FUNCTION F_Inc : BOOL
VAR_INPUT
    in : ANY_INT;
END_VAR
VAR
    pSINT  : POINTER TO SINT;
    pINT   : POINTER TO INT;
    pDINT  : POINTER TO DINT;
    pLINT  : POINTER TO LINT;
    pUSINT : POINTER TO USINT;
    pUINT  : POINTER TO UINT;
    pUDINT : POINTER TO UDINT;
    pULINT : POINTER TO ULINT;
    pBYTE  : POINTER TO BYTE;
    pWORD  : POINTER TO WORD;
    pDWORD : POINTER TO DWORD;
END_VAR

CASE in.TypeClass OF
    __SYSTEM.TYPE_CLASS.TYPE_SINT:
        pSINT  := in.pValue;
        pSint^ := pSint^ + 1;

    __SYSTEM.TYPE_CLASS.TYPE_INT:
        pINT  := in.pValue;
        pINT^ := pINT^ + 1;

    __SYSTEM.TYPE_CLASS.TYPE_DINT:
        pDINT  := in.pValue;
        pDINT^ := pDINT^ + 1;

    __SYSTEM.TYPE_CLASS.TYPE_LINT:
        pLINT  := in.pValue;
        pLINT^ := pLINT^ + 1;

    __SYSTEM.TYPE_CLASS.TYPE_USINT:
        pUSINT  := in.pValue;
        pUSINT^ := pUSINT^ + 1;

    __SYSTEM.TYPE_CLASS.TYPE_UINT:
        pUINT  := in.pValue;
        pUINT^ := pUINT^ + 1;

    __SYSTEM.TYPE_CLASS.TYPE_UDINT:
        pUDINT  := in.pValue;
        pUDINT^ := pUDINT^ + 1;

    __SYSTEM.TYPE_CLASS.TYPE_ULINT:
        pULINT  := in.pValue;
        pULINT^ := pULINT^ + 1;
		
    __SYSTEM.TYPE_CLASS.TYPE_BYTE:
        pBYTE  := in.pValue;
        pBYTE^ := pBYTE^ + 1;
		
    __SYSTEM.TYPE_CLASS.TYPE_WORD:
        pWORD  := in.pValue;
        pWORD^ := pWORD^ + 1;
		
    __SYSTEM.TYPE_CLASS.TYPE_DWORD:
        pDWORD  := in.pValue;
        pDWORD^ := pDWORD^ + 1;
		
		
END_CASE

END_FUNCTION

(* stored: Version 1.1.0.1, ProductVersion 3.1.4024.12
   POU F_Inc: Id {4439e9c9-0e51-40cb-8b1b-78607b8cb559}, SpecialFunc None *)
